RoboDK station: workstation_two_pallets.rdk

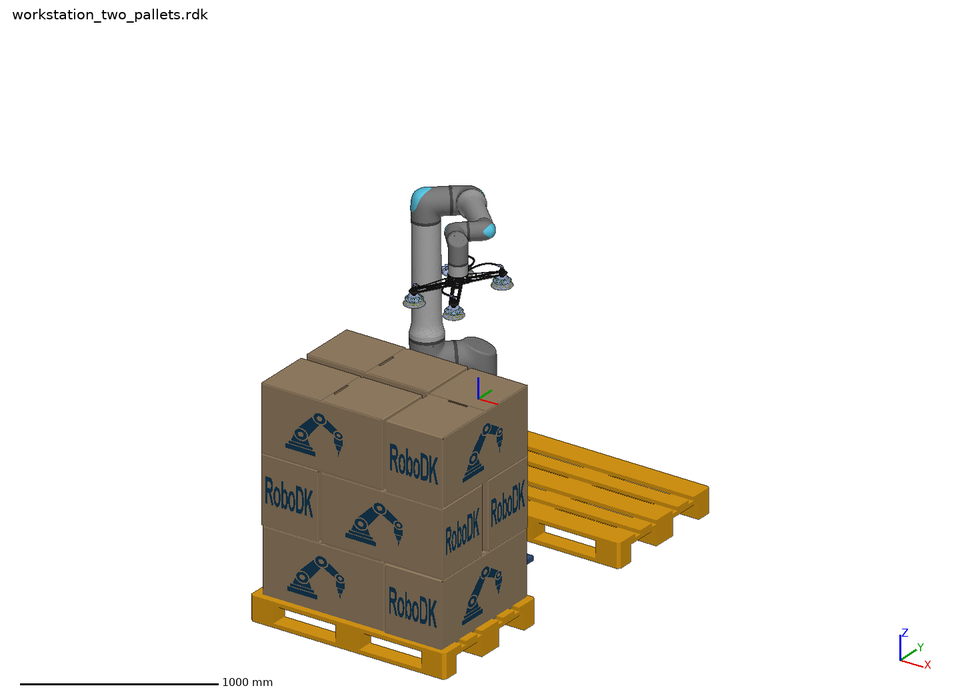
[picture v0: the station drawn from its stored meshes, robots at their saved joint values, targets as dots, program paths as lines]
Station pallet (saved by RoboDK 5.7.1). Poses are relative to the parent item; angles as X-Y-Z fixed-axis rotations.
Station parameters (name, value as stored): Box-Spawner-Settings-0
  - frame UR20 Base at (0, 0, 930) mm
    - robot UR20: 6 axes
        modified DH rows (alpha deg, a mm, theta deg, d mm): 0, 0, 0, 236.2; 90, 0, -180, 0; 0, 861.8, 0, 0; 0, 727.7, 0, 201.9; -90, 0, 0, 159.4; 90, 0, 180, 154.8
        joint limits [-360, -360, -360, -360, -360, -360] to [360, 360, 360, 360, 360, 360]; home [0, -90, -90, 0, 90, 0]; saved at [-48.257, -86.51, -80.027, -103.469, 90.117, -48.257]
      - tool PowerPick20_Large_Rectangle_20231020, TCP at (0, 0, 120) mm, size 538 x 140.6 x 358.7 mm, geometry from PowerPick20_Large_Rectangle_20231020.STEP
      - tool TOOL_FRAME, TCP at (0, 0, 120) mm
  - object EUR Pallet at (-600, 780, 0) mm, size 800 x 144 x 1200 mm, geometry from EUR Pallet.STEP
  - object Pedestal H36in (Type 1) at (0, 0, 0) mm, size 400 x 400 x 914.4 mm, geometry from Pedestal-H36in-Type-1.sld
  - object EUR Pallet at (-590, -770, 0) mm, size 800 x 144 x 1200 mm, geometry from EUR Pallet.STEP
  - object Box7 at (-540, -390, 120) mm, rotated rx 0 ry 0 rz -90 deg, size 350.3 x 751 x 400 mm, geometry from Ref_Box_MM.sld
  - object Box6 at (-540, -780, 120) mm, rotated rx 0 ry 0 rz -90 deg, size 350.3 x 751 x 400 mm, geometry from Ref_Box_MM.sld
  - object Box8 at (570, -390, 120) mm, rotated rx 0 ry 0 rz -180 deg, size 350.3 x 751 x 400 mm, geometry from Ref_Box_MM.sld
  - object Box4 at (-180, -780, 520) mm, rotated rx 0 ry 0 rz -90 deg, size 350.3 x 751 x 400 mm, geometry from Ref_Box_MM.sld
  - object Box2 at (-550, -780, 920) mm, rotated rx 0 ry 0 rz -90 deg, size 350.3 x 751 x 400 mm, geometry from Ref_Box_MM.sld
  - object Box5 at (-200, -380, 520) mm, rotated rx 0 ry 0 rz -180 deg, size 350.3 x 751 x 400 mm, geometry from Ref_Box_MM.sld
  - object Box3 at (-180, -380, 520) mm, rotated rx 0 ry 0 rz -90 deg, size 350.3 x 751 x 400 mm, geometry from Ref_Box_MM.sld
  - object Box1 at (-550, -380, 920) mm, rotated rx 0 ry 0 rz -90 deg, size 350.3 x 751 x 400 mm, geometry from Ref_Box_MM.sld
  - program ResetBoxes (9 instructions, listed below)
  - object Box0 at (570, -380, 920) mm, rotated rx 0 ry 0 rz -180 deg, size 350.3 x 751 x 400 mm, geometry from Ref_Box_MM.sld

--- program ResetBoxes (robot UR20) ---
  Replace Box0
  Replace Box1
  Replace Box2
  Replace Box3
  Replace Box4
  Replace Box5
  Replace Box6
  Replace Box7
  Replace Box8
